{attribute 'qualified_only'}
{attribute 'strict'}
TYPE E_PneumaticAxisValveState :
(
	eValveOff := 0,
	eValveOn := 1
) := eValveOff;
END_TYPE

(* stored: Version 1.1.0.1
   DUT E_PneumaticAxisValveState: Id {282877be-3966-0932-3f1c-60b7d73475d0} *)
